(* Logix 5000 project; controller AB5069L306ER_v35 vendor 1 type 14 code 196 rev 35.11; software revision 35.00 *)

MODULES
   Local : vendor 1 type 14 code 196 (5069 0, rev 35.11)
END_MODULES
